(* CoDeSys 2.3.9.35 project: PID.pro *)
(* Author: Altus *)
(* Libraries: DU35x.lib 7.7.11 15:59:13, Navigation.lib 15.7.11 10:06:00, SysLibTargetVisu.lib 26.11.08 09:53:28, Standard.lib 26.11.08 09:46:20, Iecsfc.lib 26.11.08 09:46:14, SYSLIBCALLBACK.LIB 26.11.08 09:53:30, Util.lib 26.11.08 09:46:24 *)

(* PLC configuration (modules and I/O channels)
COM1 [COM1] node 0, in %IB0 out %QB0 {BaudRate = 115200; Paridade = Sem Paridade; StopBits = 1 Stop Bit; Modem = Sem RTS/CTS; Delay = 5}
  MToolIEC [Codesys] node 0, in %IB0 out %QB0
COM2 [COM2] node 1, in %IB0 out %QB0 {BaudRate = 115200; Paridade = Sem Paridade; StopBits = 1 Stop Bit; Modem = Sem RTS/CTS; Delay = 5}
  Desabilitada [Desabilitado485] node 0, in %IB0 out %QB0
Entradas Digitais 0 [Entradas0] node 0, in %IW0 out %QB0
  I00 AT %IX0.0 [BitInput] I0.0
  I01 AT %IX0.1 [BitInput] I0.1
  I02 AT %IX0.2 [BitInput] I0.2
  I03 AT %IX0.3 [BitInput] I0.3
  I04 AT %IX0.4 [BitInput] I0.4
  I05 AT %IX0.5 [BitInput] I0.5
  I06 AT %IX0.6 [BitInput] I0.6
  I07 AT %IX0.7 [BitInput] I0.7
  I08 AT %IX0.8 [BitInput] I0.8
Entradas Digitais 1 [Entradas1] node 0, in %IW1 out %QB0
  I10 AT %IX1.0 [BitInput] I1.0
  I11 AT %IX1.1 [BitInput] I1.1
  I12 AT %IX1.2 [BitInput] I1.2
  I13 AT %IX1.3 [BitInput] I1.3
  I14 AT %IX1.4 [BitInput] I1.4
  I15 AT %IX1.5 [BitInput] I1.5
  I16 AT %IX1.6 [BitInput] I1.6
  I17 AT %IX1.7 [BitInput] I1.7
  I18 AT %IX1.8 [BitInput] I1.8
Entradas Digitais 2 [Entradas2] node 0, in %IW2 out %QB0
  I20 AT %IX2.0 [BitInput] I2.0
  I21 AT %IX2.1 [BitInput] I2.1
AI0 AT %IW4 [WordInput] AI0 {TipoAnalogica = Tensão 0-10V; FiltroAnalogica = Filtro 0 - AI=2ms  / AV=90ms; FundoEscala = 10000}
AI1 AT %IW5 [WordInput] AI1 {TipoAnalogica = Canal Desabilitado; FiltroAnalogica = Filtro 0 - AI=2ms  / AV=90ms; FundoEscala = 0}
AI2 AT %IW6 [WordInput] AI2 {TipoAnalogica = Tensão 0-10V; FiltroAnalogica = Filtro 0 - AI=2ms  / AV=90ms; FundoEscala = 10000}
AI3 AT %IW7 [WordInput] AI3 {TipoAnalogica = Channel Disable; FiltroAnalogica = Filter 0 - AI=2ms  / AV=90ms; FundoEscala = 0}
Entradas Rápidas [EntradasRapidas] node 1, in %IB16 out %QB0
  Bloco 0 [Bloco0] node 0, in %IB16 out %QB0
    Desabilitado [DesabilitadoBloco0] node 0, in %IB16 out %QB0
  Bloco 1 [Bloco1] node 1, in %IB16 out %QB0
    Desabilitado [DesabilitadoBloco1] node 0, in %IB16 out %QB0
  Entrada Configuravél Bloco 0 [EntradaConfiBloco0] node 2, in %IB16 out %QB0
    Contador 0 [EntradaConfContador0] node 0, in %IB16 out %QB0 {EntradaConfiguravelContador = Disable}
  Entrada Configuravél Bloco 1 [EntradaConfiBloco1] node 3, in %IB16 out %QB0
    Contador 2 [EntradaConfContador2] node 0, in %IB16 out %QB0 {EntradaConfiguravelContador = Disable}
Saídas Digitais 0 [Saidas0] node 0, in %IW0 out %QW0
  Q00 AT %QX0.0 [BitOutput] Q0.0
  Q01 AT %QX0.1 [BitOutput] Q0.1
  Q02 AT %QX0.2 [BitOutput] Q0.2
  Q03 AT %QX0.3 [BitOutput] Q0.3
  Q04 AT %QX0.4 [BitOutput] Q0.4
  Q05 AT %QX0.5 [BitOutput] Q0.5
  Q06 AT %QX0.6 [BitOutput] Q0.6
  Q07 AT %QX0.7 [BitOutput] Q0.7
Saídas Digitais 1 [Saidas1] node 0, in %IW0 out %QW1
  Q10 AT %QX1.0 [BitOutput] Q1.0
  Q11 AT %QX1.1 [BitOutput] Q1.1
  Q12 AT %QX1.2 [BitOutput] Q1.2
  Q13 AT %QX1.3 [BitOutput] Q1.3
  Q14 AT %QX1.4 [BitOutput] Q1.4
  Q15 AT %QX1.5 [BitOutput] Q1.5
  Q16 AT %QX1.6 [BitOutput] Q1.6
  Q17 AT %QX1.7 [BitOutput] Q1.7
AO0 AT %QW3 [WordOutput] AO0 {TipoAnalogica = Tensão 0-10V; FundoEscala = 10000}
AO1 AT %QW4 [WordOutput] AO1 {TipoAnalogica = Tensão 0-10V; FundoEscala = 10000}
Saídas Rápidas [SaidasRapidas] node 1, in %IB0 out %QB10
  Saída Rápida 0 Desabilitada [DesabilitadoF0] node 0, in %IB0 out %QB10
  Saída Rápida 1 Desabilitada [DesabilitadoF1] node 1, in %IB0 out %QB10
Saídas Comum de Contador [SaidasContador] node 2, in %IB0 out %QB10
  Saída do Bloco 0 Desabilitada [DesabilitadoSaidaBloco0] node 0, in %IB0 out %QB10
  Saída do Bloco 1 Desabilitada [DesabilitadoSaidaBloco1] node 1, in %IB0 out %QB10
Eventos Externos [Eventos] node 2, in %IB13 out %QB6
  Evento Temporizado [TimerEvent] node 0, in %IB13 out %QB6 {Intervalo = 10}
*)

(* Task configuration *)
TASK PRINCIPAL (PRIORITY := 1, INTERVAL := T#1ms);
	PLC_PRG();
END_TASK
TASK NAVIGATION (PRIORITY := 1, INTERVAL := T#20ms);
	NAVEGA();
END_TASK
TASK VISUALIZATION (PRIORITY := 1, INTERVAL := T#500ms);
	MAINTARGETVISU_PAINT_CODE
END_TASK
TASK KEYBOARD_USAGE (PRIORITY := 1, INTERVAL := T#20ms);
	MAINTARGETVISU_INPUT_CODE
END_TASK

(* POU PLC_PRG, LD *)
PROGRAM PLC_PRG
VAR
	Funcao_PID: PID;					(* Função PID *)
	Entrada_analogica: REAL;		(* Entrada da função PID que representa a entrada analógica *)
	Setpoint: REAL := 5000;				(* Setpoint -  Valor desejado *)
	Ganho_proporcional: REAL := 2;	(* Ganho Proporcional *)
	Ganho_integral: REAL := 5;		(*Redefinir o tempo, ganho de unidade recíproco da parte I; fornecido em segundos, por exemplo, "0,5" para 500 ms.*)
	Ganho_derivativo: REAL := 0.2;		(* Tempo de ação derivada, ganho de unidade da parte D em segundos, por exemplo, "0,5" para 500 ms.			*)
	Saida_manual: REAL := 4000;		(* Valor da saida do PID se entrada MANUAL estiver habilitada *)
	Offset: REAL := 0;					(* Offset para a saida Y*)
	Limite_inferior: REAL := 0;		(*Valor minimo assumido pela saída PID*)
	Limite_superior: REAL := 10000;		(*Valor máximo assumido pela saida PID*)
	Ativa_manual: BOOL := 0;			(* Ativa função PID para trabalhar em manual *)
	Reset: BOOL := 0;					(* Reseta função PID *)
	Saida_analogica: REAL := 0;		(* Saida da função PID que representa Saida analógica *)
	Limite_ativo: BOOL := 0;			(* Indica que saída da função passou os limites minimo e máximo *)
	Estouro: BOOL := 0;				(* Indica que ocorreu estouro da função. *)
END_VAR
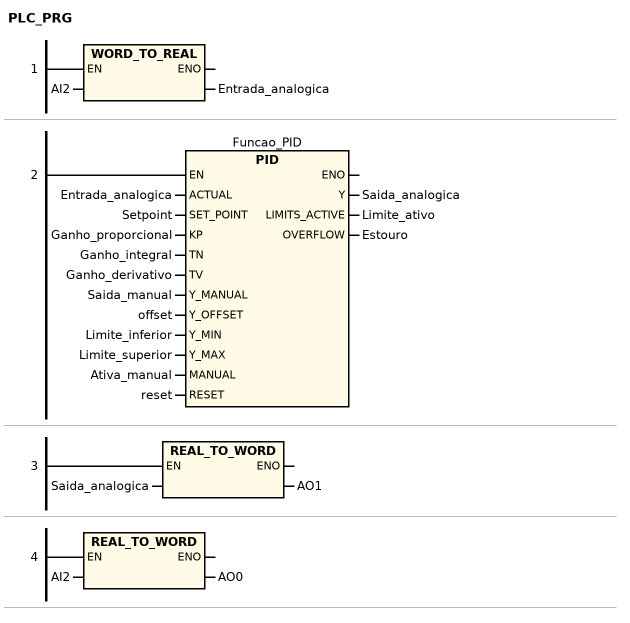
_LD_ (* Ladder Diagram *)
NETWORK 1
	*
		EN --- WORD_TO_REAL(AI2) => Entrada_analogica
NETWORK 2
	*
		EN --- Funcao_PID:PID(ACTUAL: Entrada_analogica, SET_POINT: Setpoint, KP: Ganho_proporcional, TN: Ganho_integral, TV: Ganho_derivativo, Y_MANUAL: Saida_manual, Y_OFFSET: offset, Y_MIN: Limite_inferior, Y_MAX: Limite_superior, MANUAL: Ativa_manual, RESET: reset, LIMITS_ACTIVE => Limite_ativo, OVERFLOW => Estouro) => Saida_analogica
NETWORK 3
	*
		EN --- REAL_TO_WORD(Saida_analogica) => AO1
NETWORK 4
	*
		EN --- REAL_TO_WORD(AI2) => AO0
_END_LD_
(* the same logic as Structured Text *)
(* Network 1 *)
Entrada_analogica := WORD_TO_REAL(AI2);
(* Network 2 *)
Funcao_PID(ACTUAL := Entrada_analogica, SET_POINT := Setpoint, KP := Ganho_proporcional, TN := Ganho_integral, TV := Ganho_derivativo, Y_MANUAL := Saida_manual, Y_OFFSET := offset, Y_MIN := Limite_inferior, Y_MAX := Limite_superior, MANUAL := Ativa_manual, RESET := reset);
Limite_ativo := Funcao_PID.LIMITS_ACTIVE;
Estouro := Funcao_PID.OVERFLOW;
Saida_analogica := Funcao_PID.Y;
(* Network 3 *)
AO1 := REAL_TO_WORD(Saida_analogica);
(* Network 4 *)
AO0 := REAL_TO_WORD(AI2);
END_PROGRAM

(* POU NAVEGA, ST *)
PROGRAM NAVEGA
VAR
	ControleTelas : NAVIGATION;
	ListaTelas 	: ARRAY [0..30] OF STRING(10);
END_VAR
(* Adiciona a tela MAIN como tela principal *)
ListaTelas[0] := 'MAIN';

(* Ativa o controle automático de navegação somente pelo teclado *)
ControleTelas(ENABLE_UPDW := FALSE, VISU_LIST := ListaTelas, UP := FALSE , DOWN := FALSE);
END_PROGRAM

(* Visualisation MAIN
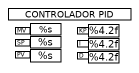
rectangle at (2,0)-(125,12): text "CONTROLADOR PID"
rectangle at (9,19)-(24,26): text "MV"
rectangle at (9,31)-(24,38): text "SP"
rectangle at (9,43)-(24,50): text "PV"
rectangle at (24,15)-(55,27): text "%s"; shows .AO1
rectangle at (71,19)-(86,26): text "KP"
rectangle at (71,32)-(86,39): text "I"
rectangle at (71,44)-(86,51): text "D"
rectangle at (24,28)-(55,40): text "%s"; shows PLC_PRG.Setpoint; editable 0..10000
rectangle at (24,41)-(55,54): text "%s"; shows .AI2
rectangle at (82,16)-(113,29): text "%4.2f"; shows PLC_PRG.Ganho_proporcional; editable 0..10000
rectangle at (82,30)-(113,42): text "%4.2f"; shows PLC_PRG.Ganho_integral; editable 0..10000
rectangle at (82,43)-(113,55): text "%4.2f"; shows PLC_PRG.Ganho_derivativo; editable 0..10000
*)
